// TIA Portal V15.1 export
// export: Created 2024-05-17T05:38:16.5840036Z, ExportSetting WithDefaults, DisplayName Totally Integrated Automation Portal, DisplayVersion V15.1 Update 5, DisplayName TIA Portal Openness, DisplayVersion V15.1 Update 5, DisplayName SINAMICS Startdrive Advanced, DisplayVersion V15.1, DisplayName G130, G150, S120, S150, SINAMICS MV, S210, DisplayVersion V15.1, DisplayName G110M, G120, G120C, G120D, G120P, DisplayVersion V15.1, DisplayName STEP 7 Professional, DisplayVersion V15.1 Update 5, DisplayName STEP 7 Safety, DisplayVersion V15.1, DisplayName WinCC Professional, DisplayVersion V15.1 Update 5, DisplayName SIMATIC Visualization Architect, DisplayVersion V15.1
DATA_BLOCK "_209210CS22ProdInfo"   // DB1625
{ S7_Optimized_Access := 'TRUE' }
VERSION : 0.1
// stored: AutoNumber false, DBAccessibleFromOPCUA true, InstanceOfName LGBProdInfo, InstanceOfType FB
"LGBProdInfo"
   // VAR_INPUT
   //    I_ConfigProdSpeed { ExternalAccessible := 'False'; ExternalVisible := 'False'; ExternalWritable := 'False'} : "ProdSpeedConfig";
   //    I_ConfigProdStartStop { ExternalAccessible := 'False'; ExternalVisible := 'False'; ExternalWritable := 'False'} : "ProdStartStopConfig";
   //    I_ConfigLineFeed { ExternalAccessible := 'False'; ExternalVisible := 'False'; ExternalWritable := 'False'} : "LineFeedConfig";
   //    I_ConfigShiftRegLine { ExternalAccessible := 'False'; ExternalVisible := 'False'; ExternalWritable := 'False'} : "ShiftRegLineConfig";
   // END_VAR
   // VAR_IN_OUT
   //    H_GBProdInfo : "H_GBProdInfo";
   // END_VAR
BEGIN
END_DATA_BLOCK
